// TIA Portal V15.1 export
// export: Created 2020-06-12T07:35:45.0537109Z, ExportSetting None, DisplayName Totally Integrated Automation Portal, DisplayVersion V15.1, DisplayName TIA Portal Openness, DisplayVersion V15.1, DisplayName STEP 7 Professional, DisplayVersion V15.1, DisplayName STEP 7 Safety, DisplayVersion V15.1, DisplayName WinCC Advanced, DisplayVersion V15.1
FUNCTION "MS_call" : Void   // FC112, FBD
TITLE = Melt stations
{ S7_Optimized_Access := 'TRUE' }
// stored: SetENOAutomatically False
BEGIN

REGION Network 1: Melt station MS1
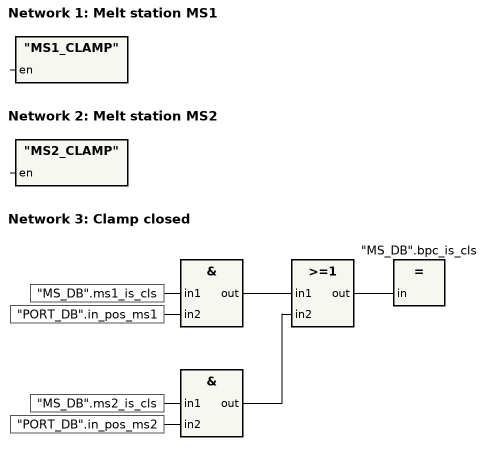
   "MS1_CLAMP"();
END_REGION

REGION Network 2: Melt station MS2
   "MS2_CLAMP"();
END_REGION

REGION Network 3: Clamp closed
   "MS_DB".bpc_is_cls := ("MS_DB".ms1_is_cls AND "PORT_DB".in_pos_ms1) OR ("MS_DB".ms2_is_cls AND "PORT_DB".in_pos_ms2);
END_REGION
END_FUNCTION
